// TIA Portal V19 export
VAR_GLOBAL   // PLC tag table "G120"
   SpeedAxis_1_Actor_Interface_AddressIn AT %I256.0 : "PD_TEL1_IN";
   SpeedAxis_1_Actor_Interface_AddressOut AT %Q256.0 : "PD_TEL1_OUT";
END_VAR
